{attribute 'GeneratedUsingTerminal: EK1122-0000-0018'}
{attribute addProperty BoxType "EK1122-0000-0018"}
{attribute addProperty Id "Beckhoff_EJx9xxsub_EK1100EK1100_AB5A94672"}
{attribute addProperty CRC "9663299"}
{attribute addProperty Size "2"}
TYPE Beckhoff_EJx9xxEK1122_00937343 EXTENDS EK1122_AB5A9467 :
STRUCT
	{attribute addProperty Name "Beckhoff_EJx9xxsub_EK1100"}
	{attribute addProperty PreviousPort "Beckhoff EJx9xxEK1122 : D"}
	Beckhoff_EJx9xxsub_EK1100 : EK1100_AB5A9467;
END_STRUCT
END_TYPE

(* stored: Version 1.2.0.0, ProductVersion 3.1.4024.9
   DUT Beckhoff_EJx9xxEK1122_00937343: Id {a58645cc-3197-4fad-9b3e-b35b2cf20c11} *)
